# EPICS substitutions: example/exampleApp/Db/userHost.substitutions
# Example substitutions file

file "db/dbExample1.db" {
    { user = "xgcHost" }
}

file db/dbExample2.db {
    pattern { user, no, scan }
        { "xgcHost", 1, "1 second" }
        { "xgcHost", 2, "2 second" }
        { "xgcHost", 3, "5 second" }
}
